TYPE ST_AxisTrqBuf :
STRUCT
	Trq  : ARRAY [0..999] OF INT;
END_STRUCT
END_TYPE

(* stored: Version 1.1.0.1, ProductVersion 3.1.4024.9
   DUT ST_AxisTrqBuf: Id {55c81aa6-67e5-45bc-9c72-6760d31724cb} *)
